// TwinCAT 3 PLC project plc_example_1
// ProgramVersion: 3.1.4023.0
// libraries:
//   lcls-twincat-motion, * (SLAC)
//   Tc2_Standard, * (Beckhoff Automation GmbH)
//   Tc2_System, * (Beckhoff Automation GmbH)
//   Tc3_Module, * (Beckhoff Automation GmbH)
// project tree:
//   / PlcTask.TcTTO
//   POUs/ MAIN.TcPOU
// real-time tasks:
//   TASK PlcTask: cycle T#10ms, priority 20, ADS port 350

CONFIGURATION plc_example_1
    RESOURCE PLC ON TwinCAT3
        TASK PlcTask(INTERVAL := T#10ms, PRIORITY := 20);
        PROGRAM MAIN WITH PlcTask : MAIN;
    END_RESOURCE
END_CONFIGURATION

// ---- POUs/MAIN.TcPOU
PROGRAM MAIN
VAR
    {attribute 'pytmc' := '
        pv: PLC:DEMO:COUNTER
    '}
    nCounter: UDINT := 10;
    sError: STRING;

    {attribute 'TcLinkTo' := 'TIIB[Term 3 (EL5042)]^FB Inputs Channel 1^Position'}
    // Special syntax for input variable
    nEncoderCount AT %I*: ULINT;
    // pragma for linking
    {attribute 'TcLinkTo' := 'TIIB[Term 6 (EL2004)]^Channel 1^Output'}
    // Special syntax for output variable
    (*
        Multi-line
        comment
    *)
    bOutput AT %Q*: BOOL;
END_VAR

nCounter := nCounter + 1;
sError := F_MotionErrorCodeLookup(nCounter);
bOutput := TRUE;

IF sError = F_MotionErrorCodeLookup(1) THEN
    nCounter := nCounter + 1;
END_IF

END_PROGRAM
